FUNCTION_BLOCK Test_TEventHandler_HandlesRaisedEvent EXTENDS T_UnitTestbase
VAR_INPUT
END_VAR
VAR_OUTPUT
END_VAR
VAR
    TestEvent : T_TestEvent;
    TestEventHandler1 : T_TestEventHandler;
    TestEventHandler2 : T_TestEventHandler;
    TestEventHandler3 : T_TestEventHandler;
    TestEventHandler4 : T_TestEventHandler;
    TestEventHandler5 : T_TestEventHandler;
END_VAR

TestEvent
    .ClearEventHandlers()
    .AddEventHandler(TestEventHandler1)
    .AddEventHandler(TestEventHandler2)
    .AddEventHandler(TestEventHandler3)
    .AddEventHandler(TestEventHandler4)
    .AddEventHandler(TestEventHandler5);
    
TestEvent.Args.Add_UDINT(21);    
TestEvent.Raise();

Assertion.AssertEquals_BOOL(
    Expected := TRUE,
    Actual   := TestEventHandler1.EventWasRaised,
    VariableName  := 'TestEventHandler1.EventWasRaised');

Assertion.AssertEquals_BOOL(
    Expected := TRUE,
    Actual   := TestEventHandler2.EventWasRaised,
    VariableName  := 'TestEventHandler2.EventWasRaised');

Assertion.AssertEquals_BOOL(
    Expected := TRUE,
    Actual   := TestEventHandler3.EventWasRaised,
    VariableName  := 'TestEventHandler3.EventWasRaised');

Assertion.AssertEquals_BOOL(
    Expected := TRUE,
    Actual   := TestEventHandler4.EventWasRaised,
    VariableName  := 'TestEventHandler4.EventWasRaised');

Assertion.AssertEquals_BOOL(
    Expected := TRUE,
    Actual   := TestEventHandler5.EventWasRaised,
    VariableName  := 'TestEventHandler5.EventWasRaised');

    
Assertion.AssertEquals_UDINT(
    Expected := 21,
    Actual   := TestEventHandler1._EventData,
    VariableName  := 'TestEventHandler1._EventData');
    
Assertion.AssertEquals_UDINT(
    Expected := 21,
    Actual   := TestEventHandler2._EventData,
    VariableName  := 'TestEventHandler2._EventData');
    
Assertion.AssertEquals_UDINT(
    Expected := 21,
    Actual   := TestEventHandler3._EventData,
    VariableName  := 'TestEventHandler3._EventData');
    
Assertion.AssertEquals_UDINT(
    Expected := 21,
    Actual   := TestEventHandler4._EventData,
    VariableName  := 'TestEventHandler4._EventData');
    
Assertion.AssertEquals_UDINT(
    Expected := 21,
    Actual   := TestEventHandler5._EventData,
    VariableName  := 'TestEventHandler5._EventData');
    
TestFinished();

END_FUNCTION_BLOCK

(* stored: Version 1.1.0.1, ProductVersion 3.1.4024.4
   POU Test_TEventHandler_HandlesRaisedEvent: Id {70af617d-87ba-4378-bd83-afa993ff0dd3}, SpecialFunc None *)
